{attribute 'qualified_only'}
VAR_GLOBAL
		//Unit rows and buttons to feedback into program
	gModeRows: typeMotionScreen;
	gModeButtons: typeMotionScreenBtn;
	
END_VAR

(* stored: Version 1.1.0.1, ProductVersion 3.1.4024.12
   GVL gModeAlternate: Id {d2a274a9-688b-442b-9dc7-7e79aecf0b90} *)
